INTERFACE INTERNAL I_TagCmp

METHOD AndIf : I_TagCmp
VAR_INPUT
	bCondition: BOOL;
END_VAR
END_METHOD

METHOD HasOption : I_TagCmp
VAR_INPUT
	sOption		: Strings.Str;
END_VAR
END_METHOD

METHOD IsErr : BOOL
END_METHOD

METHOD IsFalse : BOOL
END_METHOD

METHOD IsTrue : BOOL
END_METHOD

METHOD Match : I_TagCmp
VAR_INPUT
	iOther: I_Tag;
END_VAR
END_METHOD

METHOD MatchId : I_TagCmp
VAR_INPUT
	sIdToMatch		: Strings.Str;
END_VAR
END_METHOD

METHOD MatchWcdId : I_TagCmp
VAR_INPUT
	sPattern 			: Strings.Str;  					// Pattern with wildcards
END_VAR
END_METHOD

METHOD OrIf : I_TagCmp
VAR_INPUT
	bCondition: BOOL;
END_VAR
END_METHOD

METHOD Set : I_TagCmp
VAR_INPUT
	iBaseTag	: I_Tag;
END_VAR
END_METHOD

METHOD XorIf : I_TagCmp
VAR_INPUT
	bCondition: BOOL;
END_VAR
END_METHOD

END_INTERFACE

(* stored: Version 1.1.0.1
   Itf I_TagCmp: Id {434164ab-6703-48fd-8c7c-cbf390d14597}
   Method AndIf: Id {436de305-153d-45a1-9c24-e403a9752ee1}
   Method HasOption: Id {b84f95c7-a356-49dc-93c9-34f52a63a0d6}
   Method IsErr: Id {bdea08ea-65d7-4af4-a4f6-f3da4269e7d0}
   Method IsFalse: Id {49b183b3-7ff3-4c1f-86ad-ab7ad18768ea}
   Method IsTrue: Id {9e31c3a1-a234-461e-97b6-7c042a50360a}
   Method Match: Id {ff272183-aeae-424d-9c25-2144ef81905e}
   Method MatchId: Id {5cba49aa-7253-4bc9-829c-d83e4b3c65d2}
   Method MatchWcdId: Id {babfa847-1376-48d8-8950-170aa75af813}
   Method OrIf: Id {43b0b3b9-ad9a-4aeb-88cb-22e31aac3fe8}
   Method Set: Id {94ae1389-8107-4a7f-b005-7ced5ba44f46}
   Method XorIf: Id {d8e35498-785d-4895-9e65-30990ff7fe09} *)
